PROGRAM MAIN
VAR
	B_myByte : BYTE := 128;					// BYTE = 8 Bit Speicherplatz (0 bis 255)
	r_myReal : REAL := 0.0;			// INT = 16 Bit Speihcerplatz (-32768 bis 32767)
	ui_myUnsignedInteger : UINT := 5000;	// UINT = 16 Bit Speicherplatz (0 bis 65535)	
	w_myWord : WORD := 65535;				// WORD = 16 Bit Speicherplatz (0 bis 65535)
	b_myBool : BOOL := TRUE;				// BOOL = 8 Bit Speicherplatz
	i_valueA: REAL;
	i_valueB: REAL;
	i_myResultMinus: INT;
	l_resultFak: LINT;
	i_counterYellow : INT := 0;
	i_counterBlue : INT := 0;
END_VAR

B_myByte := 100;

//r_myReal := AdditionFunction(i_valueA := 12.43, i_valueB := 1.02);
//i_myResultMinus := SubtractionFunction(i_valueA := 200, i_valueB := 20);
DoSomeMath(r_InputA := i_valueA := 12, r_InputB := 3.4);
l_resultFak := Fakultaet(i_fakultat := 10);

IF(GVL.globButtonYellow)
	THEN
	GVL.globLightGreen := TRUE;
	i_counterYellow := i_counterYellow +1;
	CASE i_counterYellow OF
		200 : ;
		400 : ;
		600 : ;
		800 :
		1000:
		1200:
		1400:
		1600:
		1800:
		2000:
END_CASE;
ELSE
	GVL.globLightGreen := FALSE;
END_IF

IF(GVL.globButtonBlue)
	THEN
	GVL.globLightRed := TRUE;
	i_counterBlue := i_counterBlue + 1;
ELSE
	GVL.globLightRed := FALSE;
END_IF

END_PROGRAM

(* stored: Version 1.1.0.1, ProductVersion 3.1.4022.12
   POU MAIN: Id {5ae01858-891f-40dd-8569-644809c3b85e}, SpecialFunc None *)
